{attribute 'GeneratedUsingTerminal: EL3632-0000-0016'}
{attribute addProperty BoxType "EL3632-0000-0016"}
{attribute addProperty Id "Start_Time_Next_LatchAT %I*ULINT8"}
{attribute addProperty CRC "1128493506"}
{attribute addProperty Size "8"}
TYPE Next_Sync1_Time_434371C2 :
STRUCT
	{attribute addProperty Name "Start_Time_Next_Latch"}
	Start_Time_Next_Latch AT %I* : ULINT;
END_STRUCT
END_TYPE

(* stored: Version 1.2.0.0, ProductVersion 3.1.4024.9
   DUT Next_Sync1_Time_434371C2: Id {e5a7db57-7a3c-4a22-959b-c0bdf8e3dcb7} *)
